# EPICS alarm handler configuration: alh_files/mgnt_li27_lgps.alhConfig
GROUP NULL LGPS:LI27:MG01
$ALIAS LGPS
$GUIDANCE
LI27 LGPS magnets
   Group Name: LGPS:LI27:MG01
   Summary PV:  LGPS:LI27:MG01:STATSUMY
$END

GROUP LGPS:LI27:MG01  LGPS:LI27:2
CHANNEL     LGPS:LI27:2           LGPS:LI27:2:STATMSG   -----
   $FORCEPV LGPS:LI27:2:STATMSGSV -DATL 1 0
